FUNCTION_BLOCK FB_HwRef4ChHeater EXTENDS FB_CanNodeBase
VAR_INPUT
END_VAR
VAR_OUTPUT
END_VAR
VAR
	//Eingänge
	nTempActual 	AT %I* : UINT;	//aktuelle Temperatur in 1/100tel °C 
	bTempCutoff 	AT %I* : BOOL;	//Übertemperaturabschaltung wurde aktiviert
	//Ausgänge
	nPidKp 			AT %Q* : UINT; 	//PID-Reglerparameter KP
	nPidKi 			AT %Q* : UINT;	//PID-Reglerparameter KI
	nPidKd 			AT %Q* : UINT;	//PID-Reglerparameter KD
	nPidTa 			AT %Q* : USINT;	//PID-Reglerparameter TA
	bHeatingOn		AT %Q* : BOOL;	//Heizer EIN
	nTempSetpoint	AT %Q* : USINT;	//Solltemperatur in °C (ohne Kommastellen)
	bEdgeLightOn	AT %Q* : BOOL;	//Seitenlicht für Kamera EIN (nur bei Mtp)
END_VAR

IF bNodeEnabled THEN
	SUPER^();
END_IF

PROPERTY P_nPidKp : UINT
SET
nPidKp := P_nPidKp;
END_SET
GET
P_nPidKp := nPidKp;
END_GET
END_PROPERTY

PROPERTY P_nPidKd : UINT
SET
nPidKd := P_nPidKd;
END_SET
GET
P_nPidKd := nPidKd;
END_GET
END_PROPERTY

PROPERTY P_bHeatingOn : BOOL
GET
P_bHeatingOn := bHeatingOn;
END_GET
SET
bHeatingOn := P_bHeatingOn;
END_SET
END_PROPERTY

PROPERTY P_nTempSetpoint : USINT
GET
P_nTempSetpoint := nTempSetpoint;
END_GET
SET
nTempSetpoint := P_nTempSetpoint;
END_SET
END_PROPERTY

PROPERTY P_nPidKi : UINT
GET
P_nPidKi := nPidKi;
END_GET
SET
nPidKi := P_nPidKi;
END_SET
END_PROPERTY

ACTION A_ResetApp:
IF nStateA_ResetApp = 0 THEN
	fbSdoWrite(sADSNetID:= stAdsAdress.sNetId, nPortNr:= stAdsAdress.nPort,
				nIndex := cUpdateRequest.nIndex, nSubIndex := 0, nDataLength := 1, nData:= 1, bExecute:= TRUE);
	IF NOT fbSdoWrite.bBusy THEN
		IF fbSdoWrite.bError THEN
			nErrorId := fbSdoWrite.nAdsErrorId;
			nErrorId2 := fbSdoWrite.nSdoErrorId;
			nStateA_ResetApp := 99;  //Error
		ELSE
			nStateA_ResetApp := 80;
		END_IF
		fbSdoWrite(bExecute:= FALSE);
	END_IF
END_IF
END_ACTION

PROPERTY P_bTempCutoff : BOOL
GET
P_bTempCutoff := bTempCutoff;
END_GET
END_PROPERTY

PROPERTY P_bEdgeLightOn : BOOL
SET
bEdgeLightOn := P_bEdgeLightOn;
END_SET
GET
P_bEdgeLightOn := bEdgeLightOn;
END_GET
END_PROPERTY

PROPERTY P_nTempActual : UINT
GET
P_nTempActual := nTempActual;
END_GET
END_PROPERTY

PROPERTY P_nPidTa : USINT
GET
P_nPidTa := nPidTa;
END_GET
SET
nPidTa := P_nPidTa;
END_SET
END_PROPERTY

END_FUNCTION_BLOCK

(* stored: Version 1.1.0.1, ProductVersion 3.1.4020.6
   POU FB_HwRef4ChHeater: Id {f21040c9-eb65-4116-bb11-49b21cb5f021}, SpecialFunc None
   Property P_nPidKp: Id {0aa3492c-0b4c-460a-9729-9e5a9d3912d2}
   Set Set: Id {cb1fddf4-e7bf-4688-95d4-f49d460c8330}
   Get Get: Id {ebc21284-06e4-4435-a811-cb13fdf019b3}
   Property P_nPidKd: Id {1781d390-2062-48f7-adec-9e119c259598}
   Set Set: Id {2dbd15be-d2d6-45ec-9b0e-38182a764c5e}
   Get Get: Id {359cfa6b-7f0e-4f1a-9cc9-035a85511ace}
   Property P_bHeatingOn: Id {38e53cbb-f6a4-452c-86ce-70bc20f1f485}
   Get Get: Id {0827e9c5-3fb6-47f7-bb3b-103d0a1c5670}
   Set Set: Id {f77bd560-9304-40cf-b643-9059f9244aa1}
   Property P_nTempSetpoint: Id {737c3cd1-5d84-41c9-a3f2-0513585c8c29}
   Get Get: Id {487870cf-93fe-4963-b676-efacc4ee71c1}
   Set Set: Id {f4903177-8da5-4c85-8ab1-d1adc9b11056}
   Property P_nPidKi: Id {83badb2f-9b78-4182-8c0c-315d6c764e91}
   Get Get: Id {51fa2cee-cd6e-424c-8d46-00d56992d4f0}
   Set Set: Id {9157a3fe-e796-44e9-a317-4c7af96561d3}
   Action A_ResetApp: Id {aa9dbc43-ed21-47e9-a0bb-87623532fe85}
   Property P_bTempCutoff: Id {ae4db5bf-1112-4095-a6a3-e14f8a5517ea}
   Get Get: Id {408975ec-8be4-40d4-be66-feb79a43602d}
   Property P_bEdgeLightOn: Id {cda48487-0aad-496e-b7cd-7c894a26dad8}
   Set Set: Id {43bbc56a-f645-41f5-83df-473e430346f5}
   Get Get: Id {cd6602ec-3d80-4860-af07-44d56da526d4}
   Property P_nTempActual: Id {d44214d4-e442-4406-8d72-595085758188}
   Get Get: Id {aa067844-b864-40a0-a855-30f556acdd5f}
   Property P_nPidTa: Id {d7f72271-1259-49b7-9b66-a530d575f057}
   Get Get: Id {05ef108f-13ea-416f-a090-d01a7cf36bfa}
   Set Set: Id {3210af61-ab4f-4c15-b58c-00709bb519a9} *)
